       "DB_Heatbooster".AI.HBL_TT_03.fValue := "DB_Application".FromHB.DB_AI.HBL_TT_03;
       "DB_Heatbooster".AI.HBL_TT_16.fValue := "DB_Application".FromHB.DB_AI.HBL_TT_16;
       "DB_Heatbooster".AI.HBL_TT_17.fValue := "DB_Application".FromHB.DB_AI.HBL_TT_17;
       "DB_Heatbooster".AI.HBL_TT_18.fValue := "DB_Application".FromHB.DB_AI.HBL_TT_18;
       "DB_Heatbooster".AI.HBL_TT_20.fValue := "DB_Application".FromHB.DB_AI.HBL_TT_20;
       "DB_Heatbooster".AI.HBL_TT_21.fValue := "DB_Application".FromHB.DB_AI.HBL_TT_21;
       "DB_Heatbooster".AI.HBL_TT_22.fValue := "DB_Application".FromHB.DB_AI.HBL_TT_22;
       "DB_Heatbooster".AI.HBL_TT_23.fValue := "DB_Application".FromHB.DB_AI.HBL_TT_23;
       "DB_Heatbooster".AI.HBL_TT_24.fValue := "DB_Application".FromHB.DB_AI.HBL_TT_24;
       "DB_Heatbooster".AI.HBL_TT_25.fValue := "DB_Application".FromHB.DB_AI.HBL_TT_25;
       "DB_Heatbooster".AI.HBL_TT_26.fValue := "DB_Application".FromHB.DB_AI.HBL_TT_26;
       "DB_Heatbooster".AI.HBL_TT_27.fValue := "DB_Application".FromHB.DB_AI.HBL_TT_27;
       "DB_Heatbooster".AI.HBL_PT_05.fValue := "DB_Application".FromHB.DB_AI.HBL_PT_05;
       "DB_Heatbooster".AI.HBL_PT_06.fValue := "DB_Application".FromHB.DB_AI.HBL_PT_06;
       "DB_Heatbooster".AI.HBL_PT_17.fValue := "DB_Application".FromHB.DB_AI.HBL_PT_17;
       "DB_Heatbooster".AI.HBL_CT_01.fValue := "DB_Application".FromHB.DB_AI.HBL_CT_01;
       "DB_Heatbooster".AI.HBL_CT_03.fValue := "DB_Application".FromHB.DB_AI.HBL_CT_03;

       "DB_Heatbooster".AI.SSC_TT_01.fValue := "DB_Application".FromHB.DB_AI.SSC_TT_01;
       "DB_Heatbooster".AI.SSC_TT_02.fValue := "DB_Application".FromHB.DB_AI.SSC_TT_02;
       "DB_Heatbooster".AI.SSC_TT_03.fValue := "DB_Application".FromHB.DB_AI.SSC_TT_03;
       "DB_Heatbooster".AI.SSC_TT_04.fValue := "DB_Application".FromHB.DB_AI.SSC_TT_04;
       "DB_Heatbooster".AI.SSC_PIT_01.fValue := "DB_Application".FromHB.DB_AI.SSC_PIT_01;
       "DB_Heatbooster".AI.SSC_PDT_01.fValue := "DB_Application".FromHB.DB_AI.SSC_PDT_01;
       "DB_Heatbooster".AI.SSC_LT_01.fValue := "DB_Application".FromHB.DB_AI.SSC_LT_01;
   END_IF;
END_REGION

REGION Network 5 (SCL): DB_Calc
   IF #Group3Done = TRUE THEN
       "DB_Heatbooster".Calc.Compressor.CrankcaseSaturationTemperature.fValue                      := "DB_Application".FromHB.DB_Calc.Compressor_CrankcaseSaturationTemperature;
       "DB_Heatbooster".Calc.Compressor.CrankcaseSuperheat.fValue                                  := "DB_Application".FromHB.DB_Calc.Compressor_CrankcaseSuperheat;
       "DB_Heatbooster".Calc.Compressor.VolumetricEfficiency.fValue                                := "DB_Application".FromHB.DB_Calc.Compressor_VolumetricEfficiency;
       "DB_Heatbooster".Calc.Compressor.IsentropicEfficiency.fValue                                := "DB_Application".FromHB.DB_Calc.Compressor_IsentropicEfficiency;
       "DB_Heatbooster".Calc.Compressor.Massflow.fValue                                            := "DB_Application".FromHB.DB_Calc.Compressor_Massflow;

       "DB_Heatbooster".Calc.HeatSink.DeltaT.fValue                                                := "DB_Application".FromHB.DB_Calc.Heatsink_DeltaT;         
       "DB_Heatbooster".Calc.HeatSink.Pinch.fValue                                                 := "DB_Application".FromHB.DB_Calc.Heatsink_Pinch;
       "DB_Heatbooster".Calc.HeatSink.HeatRate.fValue                                              := "DB_Application".FromHB.DB_Calc.Heatsink_Heatrate;              
       "DB_Heatbooster".Calc.HeatSink.DeltaP.fValue                                                := "DB_Application".FromHB.DB_Calc.Heatsink_DeltaP;
       "DB_Heatbooster".Calc.HeatSink.Massflow.fValue                                              := "DB_Application".FromHB.DB_Calc.Heatsink_Massflow;

       "DB_Heatbooster".Calc.HeatSource.DeltaT.fValue                                              := "DB_Application".FromHB.DB_Calc.Heatsource_DeltaT;           
       "DB_Heatbooster".Calc.HeatSource.Pinch.fValue                                               := "DB_Application".FromHB.DB_Calc.Heatsource_Pinch;
       "DB_Heatbooster".Calc.HeatSource.HeatRate.fValue                                            := "DB_Application".FromHB.DB_Calc.Heatsource_Heatrate;
       "DB_Heatbooster".Calc.HeatSource.DeltaP.fValue                                              := "DB_Application".FromHB.DB_Calc.Heatsource_DeltaP;
       "DB_Heatbooster".Calc.HeatSource.Massflow.fValue                                            := "DB_Application".FromHB.DB_Calc.Heatsource_Massflow;
       "DB_Heatbooster".Calc.HeatSource.TemperatureRateOfChange.fValue                             := "DB_Application".FromHB.DB_Calc.Heatsource_TemperatureRateOfChange;

       "DB_Heatbooster".Calc.HighPressPart.CompressorSaturationTemperature.fValue                  := "DB_Application".FromHB.DB_Calc.HighPressPart_CompressorSaturationTemperature;
       "DB_Heatbooster".Calc.HighPressPart.CompressorSuperheat.fValue                              := "DB_Application".FromHB.DB_Calc.HighPressPart_CompressorSuperheat;
       "DB_Heatbooster".Calc.HighPressPart.CondenserSaturationTemperature.fValue                   := "DB_Application".FromHB.DB_Calc.HighPressPart_CondenserSaturationTemperature;
       "DB_Heatbooster".Calc.HighPressPart.CondenserSubcooling.fValue                              := "DB_Application".FromHB.DB_Calc.HighPressPart_CondenserSubcooling;
       "DB_Heatbooster".Calc.HighPressPart.ExpansionValveSubcooling.fValue                         := "DB_Application".FromHB.DB_Calc.HighPressPart_ExpansionValveSubcooling;
       "DB_Heatbooster".Calc.HighPressPart.CondenserDeltaP.fValue                                  := "DB_Application".FromHB.DB_Calc.HighPressPart_CondenserDeltaP;

       "DB_Heatbooster".Calc.LowPressPart.EvaporatorSuperheat.fValue                               := "DB_Application".FromHB.DB_Calc.LowPressPart_EvaporatorSuperheat;
       "DB_Heatbooster".Calc.LowPressPart.CompressorSuperheat.fValue                               := "DB_Application".FromHB.DB_Calc.LowPressPart_CompressorSuperheat;
       "DB_Heatbooster".Calc.LowPressPart.EvaporatorSaturationTemperature.fValue                   := "DB_Application".FromHB.DB_Calc.LowPressPart_EvaporatorSaturationTemperature;
       "DB_Heatbooster".Calc.LowPressPart.CompressorSaturationTemperature.fValue                   := "DB_Application".FromHB.DB_Calc.LowPressPart_CompressorSaturationTemperature;

       "DB_Heatbooster".Calc.System.Quality.fValue                                                 := "DB_Application".FromHB.DB_Calc.System_Quality;
       "DB_Heatbooster".Calc.System.COP.fValue                                                     := "DB_Application".FromHB.DB_Calc.System_COP;
       "DB_Heatbooster".Calc.System.ElectricalPower.fValue                                         := "DB_Application".FromHB.DB_Calc.System_ElectricalPower;
       "DB_Heatbooster".Calc.System.TemperatureLift.fValue                                         := "DB_Application".FromHB.DB_Calc.System_TemperatureLift;      
       "DB_Heatbooster".Calc.System.MotorEfficiency.fValue                                         := "DB_Application".FromHB.DB_Calc.System_MotorEfficiency;                      
       "DB_Heatbooster".Calc.System.FMEP.fValue                                                    := "DB_Application".FromHB.DB_Calc.System_FMEP;                      

       "DB_Heatbooster".Calc.Auxiliary.ShaftSealDeltaT.fValue                                      := "DB_Application".FromHB.DB_Calc.Aux_ShaftSealDeltaT;
       "DB_Heatbooster".Calc.Auxiliary.CPCPumpDeltaP.fValue                                        := "DB_Application".FromHB.DB_Calc.Aux_CPCPumpDeltaP;

       "DB_Heatbooster".Calc.Misc.EvaporatorDischargePressureMean.fValue                           := "DB_Application".FromHB.DB_Calc.Misc_EvaporatorDischargePressureMean;
       "DB_Heatbooster".Calc.Misc.EvaporatorDischargeTemperatureMin.fValue                         := "DB_Application".FromHB.DB_Calc.Misc_EvaporatorDischargeTemperatureMin;
       "DB_Heatbooster".Calc.Misc.EvaporatorDischargeTemperatureMean.fValue                        := "DB_Application".FromHB.DB_Calc.Misc_EvaporatorDischargeTemperatureMean;
       "DB_Heatbooster".Calc.Misc.OilFilterDeltaP.fValue                                           := "DB_Application".FromHB.DB_Calc.Misc_OilFilterDeltaP;
   END_IF;
END_REGION

REGION Network 6 (SCL): DB_InverterDrives & DB_Valves
   IF #Group3Done = TRUE THEN
       "DB_Heatbooster".Inverter.HBL_SC_01_A1.fValue    := "DB_Application".FromHB.DB_InverterDrives.HBL_SC_01_A1;  
       "DB_Heatbooster".Inverter.HBL_SC_01_A2.fValue    := "DB_Application".FromHB.DB_InverterDrives.HBL_SC_01_A2;  
       "DB_Heatbooster".Inverter.HBL_SC_01_A3.fValue    := "DB_Application".FromHB.DB_InverterDrives.HBL_SC_01_A3;  
       "DB_Heatbooster".Inverter.HBL_SC_02_A1.fValue    := "DB_Application".FromHB.DB_InverterDrives.HBL_SC_02_A1;  
       "DB_Heatbooster".Inverter.HBL_SC_02_A2.fValue    := "DB_Application".FromHB.DB_InverterDrives.HBL_SC_02_A2;  
       "DB_Heatbooster".Inverter.HBL_SC_02_A3.fValue    := "DB_Application".FromHB.DB_InverterDrives.HBL_SC_02_A3;  
       "DB_Heatbooster".Inverter.HBL_SC_10_A1.fValue    := "DB_Application".FromHB.DB_InverterDrives.HBL_SC_10_A1;  
       "DB_Heatbooster".Inverter.HBL_SC_10_A2.fValue    := "DB_Application".FromHB.DB_InverterDrives.HBL_SC_10_A2;  
       "DB_Heatbooster".Inverter.HBL_SC_10_A3.fValue    := "DB_Application".FromHB.DB_InverterDrives.HBL_SC_10_A3;
       "DB_Heatbooster".Inverter.HBL_SC_03_A1.fValue   := "DB_Application".FromHB.DB_InverterDrives.HBL_SC_03_A1;
       "DB_Heatbooster".Inverter.HBL_SC_03_A2.fValue   := "DB_Application".FromHB.DB_InverterDrives.HBL_SC_03_A2;
       "DB_Heatbooster".Inverter.HBL_SC_03_A3.fValue   := "DB_Application".FromHB.DB_InverterDrives.HBL_SC_03_A3;


       "DB_Heatbooster".Valve.HBL_HCV_576_A1.fValue          := "DB_Application".FromHB.DB_Valves.HBL_HCV_576_A1;  
       "DB_Heatbooster".Valve.HBL_HCV_578_A1.fValue          := "DB_Application".FromHB.DB_Valves.HBL_HCV_578_A1;
       "DB_Heatbooster".Valve.HBL_HCV_577_A1.fValue          := "DB_Application".FromHB.DB_Valves.HBL_HCV_577_A1;
       "DB_Heatbooster".Valve.HBL_HCV_579_A1.fValue          := "DB_Application".FromHB.DB_Valves.HBL_HCV_579_A1;
       "DB_Heatbooster".Valve.HBL_HCV_515_A1.fValue          := "DB_Application".FromHB.DB_Valves.HBL_HCV_515_A1;
       "DB_Heatbooster".Valve.HBL_HCV_575_A1.fValue          := "DB_Application".FromHB.DB_Valves.HBL_HCV_575_A1;
       "DB_Heatbooster".Valve.HBL_HCV_616_A1.fValue          := "DB_Application".FromHB.DB_Valves.HBL_HCV_616_A1;
       "DB_Heatbooster".Valve.HBL_HCV_700_A1.fValue          := "DB_Application".FromHB.DB_Valves.HBL_HCV_700_A1;
       "DB_Heatbooster".Valve.HBL_HCV_514_A1.fValue := "DB_Application".FromHB.DB_Valves.HBL_HCV_514_A1;
       "DB_Heatbooster".Valve.HBL_HCV_548_A1.fValue := "DB_Application".FromHB.DB_Valves.HBL_HCV_548_A1;


   END_IF;
END_REGION

REGION Network 7 (SCL): DB_DO
   IF #Group3Done = TRUE THEN
       "DB_DO".HBL_EC_01 := "DB_Application".FromHB.OilHeatersGroup1;
       "DB_DO".HBL_EC_02 := "DB_Application".FromHB.OilHeatersGroup2;
       "DB_DO".HBL_HV_630 := "DB_Application".FromHB.HBL_HV_630;
       "DB_DO".HBL_HV_631 := "DB_Application".FromHB.HBL_HV_631;
       "DB_DO".HBL_HV_860 := "DB_Application".FromHB.HBL_HV_860;
       "DB_DO".HBL_HV_861 := "DB_Application".FromHB.HBL_HV_861;
       "DB_DO".SSC_P_01  := "DB_Application".FromHB.SSC_P_01;
       "DB_DO".SSC_F_01 := "DB_Application".FromHB.SSC_F_01;
       "DB_DO".SSC_P_02  := "DB_Application".FromHB.SSC_P_02;
       "DB_DO".CPC_P_01  := "DB_Application".FromHB.CPC_P_01;
       "DB_DO".HBL_LSH_62 := "DB_Application".FromHB.HBL_LSH_62;
       "DB_DO".HBL_LSL_63 := "DB_Application".FromHB.HBL_LSL_63;
       "DB_DO".HBL_LSH_64 := "DB_Application".FromHB.HBL_LSH_64;
       "DB_DO".HBL_LSL_864 := "DB_Application".FromHB.HBL_LSL_864;
       "DB_DO".HBL_LS_632 := "DB_Application".FromHB.HBL_LS_632;
       "DB_DO".HBL_LS_633 := "DB_Application".FromHB.HBL_LS_633;

   END_IF;
END_REGION

REGION Network 8 (SCL): Mapping to HB PLC
   // Things that could/should be directly connected to the Heatbooster, but are not
   "DB_Application".ToHB.HBL_HCV_514_A1 := "DB_TestSupport".Valve.TSA_HCV_322_A1.fValue;
   "DB_Application".ToHB.HBL_HCV_548_A1 := "DB_TestSupport".Valve.TSA_HCV_370_A1.fValue;
   "DB_Application".ToHB.HBL_TT_546 := "DB_TestSupport".AI.TSA_TT_356.fValue;
   "DB_Application".ToHB.HBL_PT_547 := "DB_TestSupport".AI.TSA_PT_374.fValue;
   "DB_Application".ToHB.HBL_HCV_515_A1 := 0.0; // no such valve installed 
   "DB_Application".ToHB.HBL_TT_901 := "DB_TestSupport".AI.TSA_TT_301.fValue;
   "DB_Application".ToHB.HBL_PT_902 := "DB_TestSupport".AI.TSA_PT_300.fValue;
   "DB_Application".ToHB.HBL_TT_512 := "DB_TestSupport".AI.TSA_TT_320.fValue;
   "DB_Application".ToHB.HBL_PT_511 := "DB_TestSupport".AI.TSA_PT_321.fValue;
   "DB_Application".ToHB.HBL_PT_519 := "DB_TestSupport".AI.TSA_PT_323.fValue;
   "DB_Application".ToHB.HBL_TT_518 := "DB_TestSupport".AI.TSA_TT_324.fValue;
   "DB_Application".ToHB.LivenessCounter := UDINT_TO_UINT(#CommCycles);
END_REGION

REGION Network 9: Group 4: Put
   // no SCL statement known for Runtime: written as a call
   #_w1 := #nGroup = 4;
   IF #bEnable THEN
       #PUT_1(REQ := #_w1 AND NOT #xGroup4.%X1,   // PUT
              ID := W#16#100,
              ADDR_1 := P#DB9.DBX0.0 BYTE 80,
              SD_1 := "DB_Application".ToHB);
   END_IF;
   #Group4Timeout(IN := #_w1, PT := #GroupTimeout);   // TON
   IF #PUT_1.DONE THEN #xGroup4.%X1 := TRUE; END_IF;
   #Group4Done := #xGroup4.%X1 OR #Group4Timeout.Q;
   IF #Group4Done THEN
       #nGroup := 1;
       #xGroup4 := 0;
       #CommCycles := #CommCycles + 1;
       #RuntimeElapsed := Runtime(mem := #RuntimeMemory);
   END_IF;
END_REGION
END_FUNCTION_BLOCK

FUNCTION "ScaleIn" : Real
{ S7_Optimized_Access := 'TRUE' }
VERSION : 0.1
   VAR_INPUT 
      nIn : Int;
   END_VAR

   VAR CONSTANT 
      f : Real := 10.0;
   END_VAR


BEGIN
	// ScaleIn
	// Convert input values in scaled INT format to REAL
	// Fixed scaling
	// 
	
	// received value INT eg 32767 -> REAL value 3276.7
	// 
	#ScaleIn := INT_TO_REAL(#nIn) / #f;
END_FUNCTION

FUNCTION "ScaleOut" : Int
{ S7_Optimized_Access := 'TRUE' }
VERSION : 0.1
   VAR_INPUT 
      fIn : Real;
   END_VAR

   VAR CONSTANT 
      f : Real := 10.0;
   END_VAR


BEGIN
	// ScaleOut
	// Scale output values from REAL to INT
	// Fixed scaling
	// 
	
	// sent value REAL eg 101.7 -> INT 1017
	// 
	#ScaleOut := REAL_TO_INT(#fIn * #f);
END_FUNCTION

FUNCTION "NaN" : Real
{ S7_Optimized_Access := 'TRUE' }
VERSION : 0.1
   VAR CONSTANT 
      nan : Real := 16#7FC0_0000;
   END_VAR


BEGIN
	// Note: nan is defined as a REAL constant first, else the return statement interprets 16#7FC0_0000 as a UDINT literal and converts it to REAL
	// This will always result in a valid value, and not NaN. Gotcha!
	#Ret_Val := #nan;
	
END_FUNCTION

DATA_BLOCK "InputProcessing_DB"   // DB16
AUTHOR : Heaten
VERSION : 0.1
// stored: AutoNumber true, DBAccessibleFromOPCUA true, InstanceOfName InputProcessing, InstanceOfType FB
"InputProcessing"
BEGIN
END_DATA_BLOCK

DATA_BLOCK "Cloud_DB"   // DB15
VERSION : 0.1
// stored: AutoNumber true, DBAccessibleFromOPCUA true, InstanceOfName Cloud, InstanceOfType FB
"Cloud"
BEGIN
END_DATA_BLOCK

DATA_BLOCK "Customer_DB"   // DB11
AUTHOR : Heaten
VERSION : 0.1
// stored: AutoNumber true, DBAccessibleFromOPCUA true, InstanceOfName Customer, InstanceOfType FB
"Customer"
BEGIN
END_DATA_BLOCK

DATA_BLOCK "Puma_DB"   // DB4
VERSION : 0.1
// stored: AutoNumber true, DBAccessibleFromOPCUA true, InstanceOfName Puma, InstanceOfType FB
"Puma"
BEGIN
END_DATA_BLOCK

DATA_BLOCK "CAN-Communication_DB"   // DB14
VERSION : 0.1
// stored: AutoNumber false, DBAccessibleFromOPCUA true, InstanceOfName CAN-Communication, InstanceOfType FB
"CAN-Communication"
BEGIN
END_DATA_BLOCK

DATA_BLOCK "ModbusRTUMaster_DB"   // DB27
VERSION : 0.1
// stored: AutoNumber true, DBAccessibleFromOPCUA true, InstanceOfName ModbusRTUMaster, InstanceOfType FB
"ModbusRTUMaster"
BEGIN
END_DATA_BLOCK

DATA_BLOCK "S7_Internal_DB"   // DB1
VERSION : 0.1
// stored: AutoNumber false, DBAccessibleFromOPCUA true, InstanceOfName S7_Internal, InstanceOfType FB
"S7_Internal"
BEGIN
END_DATA_BLOCK

DATA_BLOCK "Modbus_Comm_Load_DB"   // DB12
// stored: AutoNumber true, DBAccessibleFromOPCUA true, InstanceOfName Modbus_Comm_Load, OfSystemLibElement Modbus_Comm_Load, OfSystemLibVersion 5.0
"Modbus_Comm_Load"
   // VAR_INPUT
   //    REQ : Bool;
   //    PORT : PORT;
   //    BAUD : UDInt;
   //    PARITY : UInt;
   //    FLOW_CTRL : UInt;
   //    RTS_ON_DLY : UInt;
   //    RTS_OFF_DLY : UInt;
   //    RESP_TO : UInt;
   // END_VAR
   // VAR_OUTPUT
   //    DONE : Bool;
   //    ERROR : Bool;
   //    STATUS : Word;
   // END_VAR
   // VAR_IN_OUT
   //    MB_DB : P2P_MB_BASE;
   // END_VAR
   // VAR
   //    ICHAR_GAP : Word;
   //    RETRIES : Word;
   //    MODE : USInt;
   //    LINE_PRE : USInt;
   //    BRK_DET : USInt;
   //    EN_DIAG_ALARM : Bool;
   //    STOP_BITS : USInt;
   //    EN_SUPPLY_VOLT : Bool;
   //    b_e_REQ : Bool;
   //    y_state : SInt;
   //    Send_Config { S7_SetPoint := 'True'} : Send_Config;
   //    Receive_Config { S7_SetPoint := 'True'} : Receive_Config;
   //    Receive_Conditions { S7_SetPoint := 'True'} : Receive_Conditions;
   //    WRREC { S7_SetPoint := 'True'} : WRREC;
   //    RDREC { S7_SetPoint := 'True'} : RDREC;
   //    port_w_record { ExternalVisible := 'False'; S7_SetPoint := 'True'} : P2P_MB_PortData;
   //    err_record { ExternalVisible := 'False'; S7_SetPoint := 'True'} : P2P_RdEstat;
   //    ftrs_w_record { ExternalVisible := 'False'; S7_SetPoint := 'True'} : P2P_FeaturesData;
   //    wlen : UInt;
   // END_VAR
BEGIN
END_DATA_BLOCK

DATA_BLOCK "Modbus_Master_DB"   // DB38
// stored: AutoNumber true, DBAccessibleFromOPCUA true, InstanceOfName Modbus_Master, OfSystemLibElement Modbus_Master, OfSystemLibVersion 5.0
"Modbus_Master"
   // VAR_INPUT
   //    REQ : Bool;
   //    MB_ADDR : UInt;
   //    MODE : USInt;
   //    DATA_ADDR : UDInt;
   //    DATA_LEN : UInt;
   // END_VAR
   // VAR_OUTPUT
   //    DONE : Bool;
   //    BUSY : Bool;
   //    ERROR : Bool;
   //    STATUS : Word;
   // END_VAR
   // VAR_IN_OUT
   //    DATA_PTR : Variant;
   // END_VAR
   // VAR
   //    MB_State : SInt;
   //    Blocked_Proc_Timeout : Real;
   //    Extended_Addressing : Bool;
   //    Compatibility_Mode : Bool;
   //    MB_DB { S7_SetPoint := 'True'} : P2P_MB_BASE;
   //    Send_P2P { S7_SetPoint := 'True'} : Send_P2P;
   //    Receive_P2P { S7_SetPoint := 'True'} : Receive_P2P;
   //    Receive_Reset { S7_SetPoint := 'True'} : Receive_Reset;
   //    S_PORT : Word;
   //    S_RESP_TO : Word;
   //    S_ICHAR_GAP : Word;
   //    S_RETRIES : Word;
   //    S_MB_ADDR : UInt;
   //    S_MODE : USInt;
   //    S_DATA_ADDR : UDInt;
   //    S_DATA_LEN : UInt;
   //    w_retries : Word;
   //    y_SlaveAddrHi : Byte;
   //    y_SlaveAddrLo : Byte;
   //    StartAddress : Word;
   //    Value : Word;
   //    y_FCode : Byte;
   //    INTERNAL_CDATA : Array[1..257] of Byte;
   //    mb_timer { S7_SetPoint := 'True'} : TON_TIME;
   //    TimeElapsed : Bool;
   // END_VAR
BEGIN
END_DATA_BLOCK

DATA_BLOCK "RDREC_GetDiagInfo"   // DB17
// stored: AutoNumber true, DBAccessibleFromOPCUA true, InstanceOfName RDREC_SFB, OfSystemLibElement RDREC, OfSystemLibVersion 1.0
"RDREC_SFB"
   // VAR_INPUT
   //    REQ : Bool;
   //    ID : HW_IO;
   //    INDEX : DInt;
   //    MLEN : UInt;
   // END_VAR
   // VAR_OUTPUT
   //    VALID : Bool;
   //    BUSY : Bool;
   //    ERROR : Bool;
   //    STATUS : DWord;
   //    LEN : UInt;
   // END_VAR
   // VAR_IN_OUT
   //    RECORD : Variant;
   // END_VAR
BEGIN
END_DATA_BLOCK
